FUNCTION_BLOCK FB_WorkerDefGrid_Delete EXTENDS FB_WorkerDefGrid

METHOD PROTECTED  Attach : BOOL
VAR_INPUT
  iCT              : I_CT;                         (*container at triggered event position*)
END_VAR
IF SUPER^.Attach(iCT:=iCT) THEN
  ;
END_IF
END_METHOD

METHOD   mJobStart
VAR_INPUT
	sJobDef	: CalmarCompPrint.I_JobDefinition;
END_VAR
END_METHOD

METHOD  mJobStop
VAR_INPUT
	sStatus	: CalmarCompPrint.I_JobStatus;
END_VAR
END_METHOD

METHOD Release : BOOL
VAR_INPUT
  iCT              : I_CT;                         (*container at triggered event position*)
END_VAR
IF SUPER^.Release(iCT := iCT) THEN
  
  // it's the last worker so distroy attached CT
  IF _pCTM <> 0 THEN
    LogLvl(Lvl:=E_LogSeverity.Debug, Msg:=F_Concat2('DestroyCT: ', TO_STRING(iCT.pCT^.iId)));
    _pCTM^.DestroyCT(iCT:=iCT);
  END_IF
  
END_IF
END_METHOD

METHOD  work
SUPER^.work();

IF _pAttachedCt <> 0 THEN
  Release(iCT:=_pAttachedCt^);
END_IF
END_METHOD

END_FUNCTION_BLOCK

(* stored: Version 1.1.0.1, ProductVersion 3.1.4024.11
   POU FB_WorkerDefGrid_Delete: Id {7527e8ae-b298-40c4-9d5c-225c5c9f33be}, SpecialFunc None
   Folder I_PrintStatusClient: Id {6e3174a4-81f1-4e18-94c7-de9c90656509}
   Method Attach: Id {ba44b2bb-b602-4351-b884-27d38546747f}
   Method mJobStart: Id {cad8a58f-798d-4ce1-b364-734a7078cd17}
   Method mJobStop: Id {e745e5b1-0639-4bb5-a186-c326d0f28306}
   Method Release: Id {7ef7389d-1596-4a7c-82f8-404606f272e5}
   Method work: Id {7026ea79-caca-4595-a7ed-707178d44865} *)
